DATA_BLOCK "AutoProcessData"
VAR
  A_ScanRotate : "ProcessData";
  F_Robot1Grip1 : "ProcessData";
  F_Robot1Grip2 : "ProcessData";
  B_Press1 : "ProcessData";
  C_Glue : "ProcessData";
  F_Robot2Grip1 : "ProcessData";
  F_Robot2Grip2 : "ProcessData";
  C_GlueNGBuffer : "ProcessData";
  C_MagnScanNGBuffer : "ProcessData";
  B_Press2 : "ProcessData";
  F_Robot3Grip1 : "ProcessData";
  F_Robot3Grip2 : "ProcessData";
  H_ShafeLine : "ProcessData";
  J_MagnetBelt : "ProcessData";
  K_ReserveBelt : "ProcessData";
  L_UnloadBelt : "ProcessData";
  ClearData : "ProcessData";
  A_Table_1 : Array[1..10] of "TableProcessData";
  A_Table_2 : Array[1..10] of "TableProcessData";
  FixtureCode_A1 : Array[1..10] of String[128];
  FixtureCode_A2 : Array[1..10] of String[128];
  GlobalData : STRUCT
    Table1CodeOKFlag : Bool;
    Table2CodeOKFlag : Bool;
    Fixture1CodeOKFlag : Bool;
    Fixture2CodeOKFlag : Bool;
    Robot2GripperCodeOKFlag : Bool;
    Robot1GripperCodeOKFlag : Bool;
    Robot3GripperCodeOKFlag : Bool;
    Spare_8 : Bool;
    Spare_9 : Bool;
    Spare_10 : Bool;
    Spare_11 : Bool;
    Spare_12 : Bool;
    Spare_13 : Bool;
    Spare_14 : Bool;
    Spare_15 : Bool;
    Spare_16 : Bool;
    DataIndex : Int;
    Robot1GripCodeStatus1 : Int;
    Robot1GripCodeStatus2 : Int;
    Robot1GripCodeStatus3 : Int;
    Robot1GripCodeStatus4 : Int;
    Robot2GripCodeStatus1 : Int;
    Robot2GripCodeStatus2 : Int;
    Robot2GripCodeStatus3 : Int;
    Robot2GripCodeStatus4 : Int;
    Robot3GripCodeStatus1 : Int;
    Robot3GripCodeStatus2 : Int;
    Robot3GripCodeStatus3 : Int;
    Robot3GripCodeStatus4 : Int;
    FixtureCode_A1Status1 : Int;
    FixtureCode_A1Status2 : Int;
    FixtureCode_A1Status3 : Int;
    FixtureCode_A1Status4 : Int;
    FixtureCode_A1Status5 : Int;
    FixtureCode_A1Status6 : Int;
    FixtureCode_A1Status7 : Int;
    FixtureCode_A1Status8 : Int;
    FixtureCode_A1Status9 : Int;
    FixtureCode_A1Status10 : Int;
    FixtureCode_A2Status1 : Int;
    FixtureCode_A2Status2 : Int;
    FixtureCode_A2Status3 : Int;
    FixtureCode_A2Status4 : Int;
    FixtureCode_A2Status5 : Int;
    FixtureCode_A2Status6 : Int;
    FixtureCode_A2Status7 : Int;
    FixtureCode_A2Status8 : Int;
    FixtureCode_A2Status9 : Int;
    FixtureCode_A2Status10 : Int;
    Spare : Array[1..332] of Byte;
  END_STRUCT;
  DataBuffer : Array[1..30] of "ProcessData";
  GripperCode_R1 : Array[1..10] of String[128];
  GripperCode_R2 : Array[1..10] of String[128];
  GripperCode_R3 : Array[1..10] of String[128];
END_VAR
BEGIN
END_DATA_BLOCK
